(* IEC 61131-3 sources: standardizer-tutorial-lib/test, 8 files *)

(* ---- UserAssert.st ---- *)
USING Simatic.Ax.Tutorial;
USING AxUnit.Assert;

NAMESPACE Simatic.Ax.UserAsserts
    // Assertions for enumerations
    FUNCTION Equal : BOOL
        VAR_INPUT
                expected: ValveState;
                actual: ValveState;
        END_VAR
        Equal := expected = actual;
    END_FUNCTION
END_NAMESPACE

(* ---- Test_Add.st ---- *)
USING Axunit;
USING Simatic.Ax.Tutorial;

NAMESPACE Siemens.Tiax.Tests

    {TestFixture}
    CLASS Test_Add

        {Test}
        METHOD PUBLIC Test_values
            VAR_TEMP
                result : DINT;
            END_VAR
            Add(v1 := 1, v2 := 1 , result => result);
            Axunit.Assert.Equal(2, result);

            Add(v1 := -1, v2 := -1 , result => result);
            Axunit.Assert.Equal(DINT#-2, result);

            Add(v1 := 1, v2 := -1 , result => result);
            Axunit.Assert.Equal(DINT#0, result);

            Add(v1 := -1, v2 := 1 , result => result);
            Axunit.Assert.Equal(DINT#0, result);
        END_METHOD
    END_CLASS

END_NAMESPACE

(* ---- Test_Valve.st ---- *)
NAMESPACE Tutorial.Test
    {TestFixture}
    CLASS TestMyValve
        VAR PRIVATE

        END_VAR

    END_CLASS
END_NAMESPACE

(* ---- TestAnalogFillingLevel.st ---- *)
USING Simatic.Ax.Tutorial;
USING Simatic.Ax.IO.Input;
USING Simatic.Ax.UserAsserts;

NAMESPACE Tutorial.Test
    {TestFixture}
    CLASS Valve_AnalogFillingLevel
        VAR PRIVATE
            v : FillingLevelAnalogValue;

        END_VAR

        {Test}
        METHOD PUBLIC SetFillingLevel_500_and_expect_500
            v.Level.ReadCyclic(value := LREAL#500.0);
            AxUnit.Assert.Equal(expected := 500.0, actual := v.GetFillingLevel());
        END_METHOD
    END_CLASS
END_NAMESPACE

(* ---- TestBaseValve.st ---- *)
USING Simatic.Ax.Tutorial;
USING Simatic.Ax.IO.Output;
USING Simatic.Ax.UserAsserts;

NAMESPACE Tutorial.Test
    {TestFixture}
    CLASS Valve_Test_Class
        VAR PRIVATE
            v : Solution.Valve;
            _qOpen : BinOutput;
        END_VAR

        {Test}
        METHOD PUBLIC Test_ctrlOpen_default_value_expect_false
            v.SetRefToDQ(_qOpen);
            AxUnit.Assert.Equal(expected := FALSE, actual := _qOpen.IsOn());
        END_METHOD

        {Test}
        METHOD PUBLIC Test_ValveClose_default_value_expect_false
            v.SetRefToDQ(_qOpen);
            v.Open();  // open it before
            v.Close();
            AxUnit.Assert.Equal(expected := FALSE, actual :=  _qOpen.IsOn());
        END_METHOD

        {Test}
        METHOD PUBLIC Test_ValveOpen_and_expect_ctrlOpen_true
            v.SetRefToDQ(_qOpen);
            v.Open();
            AxUnit.Assert.Equal(expected := TRUE, actual :=  _qOpen.IsOn());
            ;
        END_METHOD

        {Test}
        METHOD PUBLIC Test_GetStateOf_ClosedValve
            v.SetRefToDQ(_qOpen);
            AxUnit.Assert.Equal(expected := TRUE, actual := Equal(ValveState#Closed, v.GetState()));
        END_METHOD

        {Test}
        METHOD PUBLIC Test_GetStateOf_OpenedValve
            v.SetRefToDQ(_qOpen);
            v.Open();
            AxUnit.Assert.Equal(expected := TRUE, actual := Equal(ValveState#Open, v.GetState()));
        END_METHOD

    END_CLASS
END_NAMESPACE

(* ---- TestHeatBlock.st ---- *)
USING Simatic.Ax.Tutorial;

NAMESPACE Tutorial.Test
    {TestFixture}
    CLASS TestHeatBlock
        VAR PRIVATE
            _heatBlock : HeatBlock := (TemperatureSp := (Value := 80.0));
        END_VAR

        {Test}
        METHOD PUBLIC Test_GetSetpoint_Expect_80
            AxUnit.Assert.Equal(expected := 80.0, actual := _heatBlock.GetSetpoint());
        END_METHOD

        {Test}
        METHOD PUBLIC Test_SetSetpoint_120_And_Expect_120
            _heatBlock.SetSetpoint(120.0);
            AxUnit.Assert.Equal(expected := 120.0, actual := _heatBlock.GetSetpoint());

        END_METHOD

        {Test}
        METHOD PUBLIC Enable_Heatblock_expect_enabled_true
            AxUnit.Assert.Equal(expected := FALSE, actual := _heatBlock.IsEnabled());
            _heatBlock.Enable();
            AxUnit.Assert.Equal(expected := TRUE, actual := _heatBlock.IsEnabled());
            _heatBlock.Disable();
            AxUnit.Assert.Equal(expected := FALSE, actual := _heatBlock.IsEnabled());
        END_METHOD

    END_CLASS
END_NAMESPACE

(* ---- TestTank.st ---- *)
USING Simatic.Ax.Tutorial;

NAMESPACE Tutorial.Test
    {TestFixture}
    CLASS TestTank
        VAR PRIVATE
            _tank : Tank := (CapacityLiters := 500.0);
            _fl : FillingLevelConstant500Liter;
        END_VAR

        {Test}
        METHOD PUBLIC Test_GetCapacity_and_expect_500
            _tank.ConnectFillingLevel(_fl);
            AxUnit.Assert.Equal(expected := 500.0, actual := _tank.GetCapacity());
        END_METHOD

        {Test}
        METHOD PUBLIC Test_IsFull_and_expect_true
            _tank.ConnectFillingLevel(_fl);
            AxUnit.Assert.Equal(expected := TRUE, actual := _tank.IsFull());

        END_METHOD

        {Test}
        METHOD PUBLIC Test_GetFillingLevel_andExpect_500
            _tank.ConnectFillingLevel(_fl);
            AxUnit.Assert.Equal(expected := 500.0, actual := _tank.GetFillingLevel());
        END_METHOD
    END_CLASS
END_NAMESPACE

(* ---- TestValveWithClosedSensor.st ---- *)
USING Simatic.Ax.Tutorial;
USING Simatic.Ax.IO.Output;
USING Simatic.Ax.IO.Input;
USING Simatic.Ax.UserAsserts;

NAMESPACE Tutorial.Test
    {TestFixture}
    CLASS ValveFbClosed_Test_Class
        VAR PRIVATE
            v : ValveFbClosed;
            _qOpen : BinOutput;
            _fbClosed : BinSignal;
        END_VAR

        {Test}
        METHOD PUBLIC Test_ctrlOpen_default_value_expect_false
            v.SetRefToDQ(_qOpen);
            AxUnit.Assert.Equal(expected := FALSE, actual := _qOpen.IsOn());
        END_METHOD

        {Test}
        METHOD PUBLIC Test_ValveClose_default_value_expect_false
            v.SetRefToDQ(_qOpen);
            v.Open();  // open it before
            v.Close();
            AxUnit.Assert.Equal(expected := FALSE, actual := _qOpen.IsOn());
        END_METHOD

        {Test}
        METHOD PUBLIC Test_ValveOpen_and_expect_ctrlOpen_true
            v.SetRefToDQ(_qOpen);
            v.Open();
            AxUnit.Assert.Equal(expected := TRUE, actual := _qOpen.IsOn());
            ;
        END_METHOD

        {Test}
        METHOD PUBLIC Test_GetStateOf_ClosedValve
            v.SetRefToDQ(_qOpen);
            v.signalFbClosed := _fbClosed;
            _fbClosed.ReadCyclic(signal := TRUE);
            AxUnit.Assert.Equal(expected := TRUE, actual := Equal(ValveState#Closed, v.GetState()));
        END_METHOD

        {Test}
        METHOD PUBLIC Test_GetStateOf_OpenedValve
            v.SetRefToDQ(_qOpen);
            v.signalFbClosed := _fbClosed;
            _fbClosed.ReadCyclic(signal := FALSE);
            v.Open();
            AxUnit.Assert.Equal(expected := TRUE, actual := Equal(ValveState#Open, v.GetState()));
        END_METHOD

    END_CLASS
END_NAMESPACE
